INTERFACE I_Sensor

PROPERTY PUBLIC Name : T_MAXSTRING
GET
END_GET
END_PROPERTY

END_INTERFACE

(* stored: Version 1.1.0.1, ProductVersion 3.1.4024.12
   Itf I_Sensor: Id {c0a80466-b393-4eb7-a2c7-d7925ddd7a2d}
   Property Name: Id {eed5ec53-5311-4cfe-9812-98d0b5b708c1}
   Get Get: Id {3b965b43-c344-4468-8c86-4b04cce40ece} *)
